(* IEC 61131-3 sources: ahu-codesys/codesys/src/03-fan-status-proof, 1 file *)

(* ---- GVL_Fan.st ---- *)
{attribute 'qualified_only'}
VAR_GLOBAL
	FanProofSignal : BOOL;
	FanFaultAlarm : BOOL;
	FanProofTimer : TON;
END_VAR
